# EPICS autosave request: iocBoot/ioc13ida_CD_Mono_XPS/auto_settings.req
file "CARS_motor_settings.req",           P=$(P), M=m57
file "CARS_motor_settings.req",           P=$(P), M=m58
file "CARS_motor_settings.req",           P=$(P), M=m59
file "CARS_motor_settings.req",           P=$(P), M=m60
file "CARS_motor_settings.req",           P=$(P), M=m61
file "CARS_motor_settings.req",           P=$(P), M=m62
file "CARS_motor_settings.req",           P=$(P), M=m63
file "CARS_motor_settings.req",           P=$(P), M=m64
file "GSE_MonoEnergy_settings.req",       P=$(P), MONO=CDEn
file "GSE_CD_MonoPositions_settings.req", P=$(P), MONO=CDEn
file "quadEM_settings.req",               P=$(P), R=QE1:
file "quadEM_Plugin_settings.req",        P=$(P), R=QE1:
file "mono_pid_control_settings.req",     P=$(P), PID=mono_pid1
file "mono_pid_control_settings.req",     P=$(P), PID=mono_pid2
file "mono_pid_control_settings.req",     P=$(P), PID=mono_pid3
file "mono_pid_control_settings.req",     P=$(P), PID=mono_pid4
